// TIA Portal V19 export
TYPE "udt_RollformingMng_Pers"
   STRUCT
      Data : Struct
         MaterialPresence : Bool;
         MaterialPresence_Entry : Bool;
         MaterialPresence_BeforeMW : Bool;
         MaterialPresence_AfterMW : Bool;
         MatPresence_ConveyorEntry : Bool;
         FinalCut_DoneGood : Bool;
         FinalCut_DoneWrong : Bool;
         FinalCut_MemTargetResult : Bool;
         ProfileHead_Found : Bool;
         HeadingDone : Bool;
         OldPPrf_PrgNo : DInt;
         ActTarget : "udt_RollformingMng_Target";
         NextTarget : "udt_RollformingMng_Target";
         FS : Struct
            LastCut_Material_Position : LReal;
            LastJob_Material_Position : LReal;
            PrevCut_Material_Position : LReal;
            PrevJob_Material_Position : LReal;
         END_STRUCT;
         CutLenght : Struct
            CarriageMeasID { ExternalAccessible := 'False'; ExternalVisible := 'False'; ExternalWritable := 'False'} : UInt;
            WheelMeasID { ExternalAccessible := 'False'; ExternalVisible := 'False'; ExternalWritable := 'False'} : UInt;
            CarriageEncoder { ExternalAccessible := 'False'; ExternalVisible := 'False'; ExternalWritable := 'False'} : LReal;
            WheelEncoder { ExternalAccessible := 'False'; ExternalVisible := 'False'; ExternalWritable := 'False'} : LReal;
            LastCut_Material_Position { ExternalAccessible := 'False'; ExternalVisible := 'False'; ExternalWritable := 'False'} : LReal;
            PrevCut_Material_Position { ExternalAccessible := 'False'; ExternalVisible := 'False'; ExternalWritable := 'False'} : LReal;
         END_STRUCT;
      END_STRUCT;
      Par : Struct
         Override : Struct
            ProductionRateOverride : LReal;
            ChangeRateStepPercentage : LReal;
            EarlyPieces_Qty : Int;
            EarlyPieces_Percentage : LReal;
            Emptying_Percentage : LReal;
            ProdSlowDow_Percentage : LReal;
            WeldPieces_Qty : Int;
            WeldSlowDow_Percentage : LReal;
            AccRollSlowDown_Percentage : LReal;
         END_STRUCT;
         SemiAut : Struct
            Enable : Bool;
            Vel : LReal;
            Acc : LReal;
            Dec : LReal;
            Jerk : LReal;
         END_STRUCT;
         TimeStopInactivity : Time := T#1M;
         AutoHeadingDistance { ExternalAccessible := 'False'; ExternalVisible := 'False'; ExternalWritable := 'False'} : LReal := 2000.0;   // Position of profile head relative to the zero position of the carriage
         ExtractionDistance { ExternalAccessible := 'False'; ExternalVisible := 'False'; ExternalWritable := 'False'} : LReal := 550.0;   // Gap between cutoff position and extractor pinch-roll
         AccRollsDistanceFromZero : LReal := 1500.0;   // Gap from zero position of the carriage to sensor entry of rolway
      END_STRUCT;
   END_STRUCT;
END_TYPE
